// TIA Portal V15.1 export
// export: Created 2020-12-23T11:16:33.2864918Z, ExportSetting WithDefaults, WithReadOnly, DisplayName Totally Integrated Automation Portal, DisplayVersion V15.1 Update 3, DisplayName TIA Portal Openness, DisplayVersion V15.1, DisplayName STEP 7 Professional, DisplayVersion V15.1 Update 3, DisplayName WinCC Advanced, DisplayVersion V15.1 Update 3
DATA_BLOCK "DBVALVES"   // DB1330
{ S7_Optimized_Access := 'TRUE' }
VERSION : 0.1
// stored: AutoNumber false, CodeModifiedDate 2020-12-23T11:16:22.2079236Z, CompileDate 2020-12-23T11:16:23.5925798Z, CreationDate 2020-12-23T11:14:57.9258238Z, DBAccessibleFromOPCUA true, DownloadWithoutReinit false, InterfaceModifiedDate 2020-12-23T11:16:22.2079236Z, IsConsistent true, IsKnowHowProtected false, IsOnlyStoredInLoadMemory false, IsPLCDB false, IsRetainMemResEnabled false, IsWriteProtectedInAS false, MemoryReserve 100, ModifiedDate 2020-12-23T11:16:22.2079236Z, ParameterModified 2020-12-23T11:16:22.2079236Z, StructureModified 2020-12-23T11:16:22.2079236Z
   VAR
      "TBL TABLE LH" : "3state";   // [1] TBL TABLE LH
      "TBL TABLE RH" : "3state";   // [2] TBL TABLE RH
      "TBL SECTION1" : "3state";   // [3] TBL SECTION1
      "TBL SECTION2" : "3state";   // [4] TBL SECTION2
      "TBL SECTION4 LH" : "3state";   // [5] TBL SECTION4 LH
      "TBL SECTION4 RH" : "3state";   // [6] TBL SECTION4 RH
      "TBL SECTION5 LH" : "3state";   // [7] TBL SECTION5 LH
      "TBL SECTION5 RH" : "3state";   // [8] TBL SECTION5 RH
      "TBL POSITIONING LH" : "3state";   // [9] TBL POSITIONING LH
      "TBL POSITIONING RH" : "3state";   // [10] TBL POSITIONING RH
      "TBL PIN LH" : "3state";   // [11] TBL PIN LH
      "TBL PIN RH" : "3state";   // [12] TBL PIN RH
      "TBL SCREW GRIPPER" : "3state";   // [13] TBL SCREW GRIPPER
      "TBL WRAP GRIPPER" : "3state";   // [14] TBL WRAP GRIPPER
      "ST1 POSITIONING" : "3state";   // [15] ST1 POSITIONING
      "ST1 SWORD" : "3state";   // [16] ST1 SWORD
      "ST2 POSITIONING" : "3state";   // [17] ST2 POSITIONING
      "ST2 SWORD" : "3state";   // [18] ST2 SWORD
      "ST3 POSITIONING" : "3state";   // [19] ST3 POSITIONING
      "ST3 SWORD A SQUEEZING" : "3state";   // [20] ST3 SWORD A SQUEEZING
      "ST3 SWORD A SPREADING" : "3state";   // [21] ST3 SWORD A SPREADING
      "ST3 SWORD A OPENING" : "3state";   // [22] ST3 SWORD A OPENING
      "ST3 SWORD B SQUEEZING" : "3state";   // [23] ST3 SWORD B SQUEEZING
      "ST3 SWORD B SPREADING" : "3state";   // [24] ST3 SWORD B SPREADING
      "ST3 SWORD B OPENING" : "3state";   // [25] ST3 SWORD B OPENING
      "ST6 CONNECTOR1" : "3state";   // [26] ST6 CONNECTOR1
      "ST6 CONNECTOR2" : "3state";   // [27] ST6 CONNECTOR2
      "ST6 HOLDFAST LH1" : "3state";   // [28] ST6 HOLDFAST LH1
      "ST6 HOLDFAST LH2" : "3state";   // [29] ST6 HOLDFAST LH2
      "ST6 HOLDFAST RH1" : "3state";   // [30] ST6 HOLDFAST RH1
      "ST6 HOLDFAST RH2" : "3state";   // [31] ST6 HOLDFAST RH2
      "ST6 ROTATION LH" : "3state";   // [32] ST6 ROTATION LH
      "ST6 ROTATION RH" : "3state";   // [33] ST6 ROTATION RH
   END_VAR
BEGIN
   // "TBL TABLE LH".in : [1] TBL TABLE LH
   // "TBL TABLE LH".in.move_hp : [1] TBL TABLE LH
   // "TBL TABLE LH".in.move_wp : [1] TBL TABLE LH
   // "TBL TABLE LH".in.move_idle : [1] TBL TABLE LH
   // "TBL TABLE LH".out : [1] TBL TABLE LH
   // "TBL TABLE RH".in : [2] TBL TABLE RH
   // "TBL TABLE RH".in.move_hp : [2] TBL TABLE RH
   // "TBL TABLE RH".in.move_wp : [2] TBL TABLE RH
   // "TBL TABLE RH".in.move_idle : [2] TBL TABLE RH
   // "TBL TABLE RH".out : [2] TBL TABLE RH
   // "TBL SECTION1".in : [3] TBL SECTION1
   // "TBL SECTION1".in.move_hp : [3] TBL SECTION1
   // "TBL SECTION1".in.move_wp : [3] TBL SECTION1
   // "TBL SECTION1".in.move_idle : [3] TBL SECTION1
   // "TBL SECTION1".out : [3] TBL SECTION1
   // "TBL SECTION2".in : [4] TBL SECTION2
   // "TBL SECTION2".in.move_hp : [4] TBL SECTION2
   // "TBL SECTION2".in.move_wp : [4] TBL SECTION2
   // "TBL SECTION2".in.move_idle : [4] TBL SECTION2
   // "TBL SECTION2".out : [4] TBL SECTION2
   // "TBL SECTION4 LH".in : [5] TBL SECTION4 LH
   // "TBL SECTION4 LH".in.move_hp : [5] TBL SECTION4 LH
   // "TBL SECTION4 LH".in.move_wp : [5] TBL SECTION4 LH
   // "TBL SECTION4 LH".in.move_idle : [5] TBL SECTION4 LH
   // "TBL SECTION4 LH".out : [5] TBL SECTION4 LH
   // "TBL SECTION4 RH".in : [6] TBL SECTION4 RH
   // "TBL SECTION4 RH".in.move_hp : [6] TBL SECTION4 RH
   // "TBL SECTION4 RH".in.move_wp : [6] TBL SECTION4 RH
   // "TBL SECTION4 RH".in.move_idle : [6] TBL SECTION4 RH
   // "TBL SECTION4 RH".out : [6] TBL SECTION4 RH
   // "TBL SECTION5 LH".in : [7] TBL SECTION5 LH
   // "TBL SECTION5 LH".in.move_hp : [7] TBL SECTION5 LH
   // "TBL SECTION5 LH".in.move_wp : [7] TBL SECTION5 LH
   // "TBL SECTION5 LH".in.move_idle : [7] TBL SECTION5 LH
   // "TBL SECTION5 LH".out : [7] TBL SECTION5 LH
   // "TBL SECTION5 RH".in : [8] TBL SECTION5 RH
   // "TBL SECTION5 RH".in.move_hp : [8] TBL SECTION5 RH
   // "TBL SECTION5 RH".in.move_wp : [8] TBL SECTION5 RH
   // "TBL SECTION5 RH".in.move_idle : [8] TBL SECTION5 RH
   // "TBL SECTION5 RH".out : [8] TBL SECTION5 RH
   // "TBL POSITIONING LH".in : [9] TBL POSITIONING LH
   // "TBL POSITIONING LH".in.move_hp : [9] TBL POSITIONING LH
   // "TBL POSITIONING LH".in.move_wp : [9] TBL POSITIONING LH
   // "TBL POSITIONING LH".in.move_idle : [9] TBL POSITIONING LH
   // "TBL POSITIONING LH".out : [9] TBL POSITIONING LH
   // "TBL POSITIONING RH".in : [10] TBL POSITIONING RH
   // "TBL POSITIONING RH".in.move_hp : [10] TBL POSITIONING RH
   // "TBL POSITIONING RH".in.move_wp : [10] TBL POSITIONING RH
   // "TBL POSITIONING RH".in.move_idle : [10] TBL POSITIONING RH
   // "TBL POSITIONING RH".out : [10] TBL POSITIONING RH
   // "TBL PIN LH".in : [11] TBL PIN LH
   // "TBL PIN LH".in.move_hp : [11] TBL PIN LH
   // "TBL PIN LH".in.move_wp : [11] TBL PIN LH
   // "TBL PIN LH".in.move_idle : [11] TBL PIN LH
   // "TBL PIN LH".out : [11] TBL PIN LH
   // "TBL PIN RH".in : [12] TBL PIN RH
   // "TBL PIN RH".in.move_hp : [12] TBL PIN RH
   // "TBL PIN RH".in.move_wp : [12] TBL PIN RH
   // "TBL PIN RH".in.move_idle : [12] TBL PIN RH
   // "TBL PIN RH".out : [12] TBL PIN RH
   // "TBL SCREW GRIPPER".in : [13] TBL SCREW GRIPPER
   // "TBL SCREW GRIPPER".in.move_hp : [13] TBL SCREW GRIPPER
   // "TBL SCREW GRIPPER".in.move_wp : [13] TBL SCREW GRIPPER
   // "TBL SCREW GRIPPER".in.move_idle : [13] TBL SCREW GRIPPER
   // "TBL SCREW GRIPPER".out : [13] TBL SCREW GRIPPER
   // "TBL WRAP GRIPPER".in : [14] TBL WRAP GRIPPER
   // "TBL WRAP GRIPPER".in.move_hp : [14] TBL WRAP GRIPPER
   // "TBL WRAP GRIPPER".in.move_wp : [14] TBL WRAP GRIPPER
   // "TBL WRAP GRIPPER".in.move_idle : [14] TBL WRAP GRIPPER
   // "TBL WRAP GRIPPER".out : [14] TBL WRAP GRIPPER
   // "ST1 POSITIONING".in : [15] ST1 POSITIONING
   // "ST1 POSITIONING".in.move_hp : [15] ST1 POSITIONING
   // "ST1 POSITIONING".in.move_wp : [15] ST1 POSITIONING
   // "ST1 POSITIONING".in.move_idle : [15] ST1 POSITIONING
   // "ST1 POSITIONING".out : [15] ST1 POSITIONING
   // "ST1 SWORD".in : [16] ST1 SWORD
   // "ST1 SWORD".in.move_hp : [16] ST1 SWORD
   // "ST1 SWORD".in.move_wp : [16] ST1 SWORD
   // "ST1 SWORD".in.move_idle : [16] ST1 SWORD
   // "ST1 SWORD".out : [16] ST1 SWORD
   // "ST2 POSITIONING".in : [17] ST2 POSITIONING
   // "ST2 POSITIONING".in.move_hp : [17] ST2 POSITIONING
   // "ST2 POSITIONING".in.move_wp : [17] ST2 POSITIONING
   // "ST2 POSITIONING".in.move_idle : [17] ST2 POSITIONING
   // "ST2 POSITIONING".out : [17] ST2 POSITIONING
   // "ST2 SWORD".in : [18] ST2 SWORD
   // "ST2 SWORD".in.move_hp : [18] ST2 SWORD
   // "ST2 SWORD".in.move_wp : [18] ST2 SWORD
   // "ST2 SWORD".in.move_idle : [18] ST2 SWORD
   // "ST2 SWORD".out : [18] ST2 SWORD
   // "ST3 POSITIONING".in : [19] ST3 POSITIONING
   // "ST3 POSITIONING".in.move_hp : [19] ST3 POSITIONING
   // "ST3 POSITIONING".in.move_wp : [19] ST3 POSITIONING
   // "ST3 POSITIONING".in.move_idle : [19] ST3 POSITIONING
   // "ST3 POSITIONING".out : [19] ST3 POSITIONING
   // "ST3 SWORD A SQUEEZING".in : [20] ST3 SWORD A SQUEEZING
   // "ST3 SWORD A SQUEEZING".in.move_hp : [20] ST3 SWORD A SQUEEZING
   // "ST3 SWORD A SQUEEZING".in.move_wp : [20] ST3 SWORD A SQUEEZING
   // "ST3 SWORD A SQUEEZING".in.move_idle : [20] ST3 SWORD A SQUEEZING
   // "ST3 SWORD A SQUEEZING".out : [20] ST3 SWORD A SQUEEZING
   // "ST3 SWORD A SPREADING".in : [21] ST3 SWORD A SPREADING
   // "ST3 SWORD A SPREADING".in.move_hp : [21] ST3 SWORD A SPREADING
   // "ST3 SWORD A SPREADING".in.move_wp : [21] ST3 SWORD A SPREADING
   // "ST3 SWORD A SPREADING".in.move_idle : [21] ST3 SWORD A SPREADING
   // "ST3 SWORD A SPREADING".out : [21] ST3 SWORD A SPREADING
   // "ST3 SWORD A OPENING".in : [22] ST3 SWORD A OPENING
   // "ST3 SWORD A OPENING".in.move_hp : [22] ST3 SWORD A OPENING
   // "ST3 SWORD A OPENING".in.move_wp : [22] ST3 SWORD A OPENING
   // "ST3 SWORD A OPENING".in.move_idle : [22] ST3 SWORD A OPENING
   // "ST3 SWORD A OPENING".out : [22] ST3 SWORD A OPENING
   // "ST3 SWORD B SQUEEZING".in : [23] ST3 SWORD B SQUEEZING
   // "ST3 SWORD B SQUEEZING".in.move_hp : [23] ST3 SWORD B SQUEEZING
   // "ST3 SWORD B SQUEEZING".in.move_wp : [23] ST3 SWORD B SQUEEZING
   // "ST3 SWORD B SQUEEZING".in.move_idle : [23] ST3 SWORD B SQUEEZING
   // "ST3 SWORD B SQUEEZING".out : [23] ST3 SWORD B SQUEEZING
   // "ST3 SWORD B SPREADING".in : [24] ST3 SWORD B SPREADING
   // "ST3 SWORD B SPREADING".in.move_hp : [24] ST3 SWORD B SPREADING
   // "ST3 SWORD B SPREADING".in.move_wp : [24] ST3 SWORD B SPREADING
   // "ST3 SWORD B SPREADING".in.move_idle : [24] ST3 SWORD B SPREADING
   // "ST3 SWORD B SPREADING".out : [24] ST3 SWORD B SPREADING
   // "ST3 SWORD B OPENING".in : [25] ST3 SWORD B OPENING
   // "ST3 SWORD B OPENING".in.move_hp : [25] ST3 SWORD B OPENING
   // "ST3 SWORD B OPENING".in.move_wp : [25] ST3 SWORD B OPENING
   // "ST3 SWORD B OPENING".in.move_idle : [25] ST3 SWORD B OPENING
   // "ST3 SWORD B OPENING".out : [25] ST3 SWORD B OPENING
   // "ST6 CONNECTOR1".in : [26] ST6 CONNECTOR1
   // "ST6 CONNECTOR1".in.move_hp : [26] ST6 CONNECTOR1
   // "ST6 CONNECTOR1".in.move_wp : [26] ST6 CONNECTOR1
   // "ST6 CONNECTOR1".in.move_idle : [26] ST6 CONNECTOR1
   // "ST6 CONNECTOR1".out : [26] ST6 CONNECTOR1
   // "ST6 CONNECTOR2".in : [27] ST6 CONNECTOR2
   // "ST6 CONNECTOR2".in.move_hp : [27] ST6 CONNECTOR2
   // "ST6 CONNECTOR2".in.move_wp : [27] ST6 CONNECTOR2
   // "ST6 CONNECTOR2".in.move_idle : [27] ST6 CONNECTOR2
   // "ST6 CONNECTOR2".out : [27] ST6 CONNECTOR2
   // "ST6 HOLDFAST LH1".in : [28] ST6 HOLDFAST LH1
   // "ST6 HOLDFAST LH1".in.move_hp : [28] ST6 HOLDFAST LH1
   // "ST6 HOLDFAST LH1".in.move_wp : [28] ST6 HOLDFAST LH1
   // "ST6 HOLDFAST LH1".in.move_idle : [28] ST6 HOLDFAST LH1
   // "ST6 HOLDFAST LH1".out : [28] ST6 HOLDFAST LH1
   // "ST6 HOLDFAST LH2".in : [29] ST6 HOLDFAST LH2
   // "ST6 HOLDFAST LH2".in.move_hp : [29] ST6 HOLDFAST LH2
   // "ST6 HOLDFAST LH2".in.move_wp : [29] ST6 HOLDFAST LH2
   // "ST6 HOLDFAST LH2".in.move_idle : [29] ST6 HOLDFAST LH2
   // "ST6 HOLDFAST LH2".out : [29] ST6 HOLDFAST LH2
   // "ST6 HOLDFAST RH1".in : [30] ST6 HOLDFAST RH1
   // "ST6 HOLDFAST RH1".in.move_hp : [30] ST6 HOLDFAST RH1
   // "ST6 HOLDFAST RH1".in.move_wp : [30] ST6 HOLDFAST RH1
   // "ST6 HOLDFAST RH1".in.move_idle : [30] ST6 HOLDFAST RH1
   // "ST6 HOLDFAST RH1".out : [30] ST6 HOLDFAST RH1
   // "ST6 HOLDFAST RH2".in : [31] ST6 HOLDFAST RH2
   // "ST6 HOLDFAST RH2".in.move_hp : [31] ST6 HOLDFAST RH2
   // "ST6 HOLDFAST RH2".in.move_wp : [31] ST6 HOLDFAST RH2
   // "ST6 HOLDFAST RH2".in.move_idle : [31] ST6 HOLDFAST RH2
   // "ST6 HOLDFAST RH2".out : [31] ST6 HOLDFAST RH2
   // "ST6 ROTATION LH".in : [32] ST6 ROTATION LH
   // "ST6 ROTATION LH".in.move_hp : [32] ST6 ROTATION LH
   // "ST6 ROTATION LH".in.move_wp : [32] ST6 ROTATION LH
   // "ST6 ROTATION LH".in.move_idle : [32] ST6 ROTATION LH
   // "ST6 ROTATION LH".out : [32] ST6 ROTATION LH
   // "ST6 ROTATION RH".in : [33] ST6 ROTATION RH
   // "ST6 ROTATION RH".in.move_hp : [33] ST6 ROTATION RH
   // "ST6 ROTATION RH".in.move_wp : [33] ST6 ROTATION RH
   // "ST6 ROTATION RH".in.move_idle : [33] ST6 ROTATION RH
   // "ST6 ROTATION RH".out : [33] ST6 ROTATION RH
END_DATA_BLOCK
